TYPE "ValveMachine_COut"
VERSION : 0.1
// Block: ValveMachine_COut
   STRUCT
      CtrlSafe : Bool;
      Standstill : Bool;
      ReqOilPressure : Bool;
      Rest_CheckNext : Bool;
      Work_CheckNext : Bool;
      Rest : Bool;
      Work : Bool;
   END_STRUCT;

END_TYPE
